PROGRAM MAIN
VAR
	//stThisIsOurFirstInstanceOfAstructure : ST_Event;	
	bBoolean : BOOL := FALSE;
	
	eEventType1 : E_EventType := E_EventType.Alarm;
	eEventSeverity1 : TcEventSeverity := TcEventSeverity.Error ;
	nEventIdentity1 : UDINT := 42;
	sEventText1 : STRING (255) := 'This is a scary event';
	
	CSVPersitentEventStorage : FB_CSVPersistentEventStorage;
	EventLogger : EventLogger (CSVPersitentEventStorage);
	
END_VAR

(*
IF NOT bBoolean THEN
	UpdateEventTimeStampWithSystemTime(stEvent := stThisIsOurFirstInstanceOfAstructure);
	bBoolean := TRUE;
END_IF 
*)

IF bBoolean THEN
	EventLogger.AddEvent (eEventType1, eEventSeverity1, nEventIdentity1, sEventText1);
	bBoolean := FALSE;	
END_IF

CSVPersitentEventStorage ();

END_PROGRAM

(* stored: Version 1.1.0.1, ProductVersion 3.1.4024.12
   POU MAIN: Id {e98ae1f1-7f18-4f84-aa16-6124f5dd1075}, SpecialFunc None *)
